FUNCTION_BLOCK FB_Krajalnica_Komunikacja EXTENDS FB_LogowanieBledow_ElementZlozony
VAR_INPUT
END_VAR
VAR_OUTPUT
END_VAR
VAR
END_VAR

METHOD DefinicjaTabeliZdarzen_1031_Niemiecki : BOOL
VAR_INPUT
	arrTablicaDefinicjiZdarzenOpis			: REFERENCE TO ARRAY [1..GVL_LogowanieBledow_Stale.MAX_ILOSC_ZDARZEN] OF DUT_LogowanieBledow_ZdarzenieOpis;

END_VAR
//arrTablicaDefinicjiZdarzenOpis [iStartId+0].sOpis	:= 'DE - TESTOWA WIADOMOSC';
END_METHOD

METHOD DefinicjaTabeliZdarzen_1033_Angielski : BOOL
VAR_INPUT
	arrTablicaDefinicjiZdarzenOpis			: REFERENCE TO ARRAY [1..GVL_LogowanieBledow_Stale.MAX_ILOSC_ZDARZEN] OF DUT_LogowanieBledow_ZdarzenieOpis;

END_VAR
//arrTablicaDefinicjiZdarzenOpis [iStartId+0].sOpis	:= 'EN - TESTOWA WIADOMOSC';
END_METHOD

METHOD DefinicjaTabeliZdarzen_1045_Polski : BOOL
VAR_INPUT
	arrTablicaDefinicjiZdarzenOpis			: REFERENCE TO ARRAY [1..GVL_LogowanieBledow_Stale.MAX_ILOSC_ZDARZEN] OF DUT_LogowanieBledow_ZdarzenieOpis;

END_VAR
//arrTablicaDefinicjiZdarzenOpis [iStartId+0].sOpis	:= 'PL - TESTOWA WIADOMOSC';
END_METHOD

METHOD DefinicjaTabeliZdarzen_Ogolna : BOOL
VAR_INPUT
	arrTablicaDefinicjiZdarzen				: REFERENCE TO ARRAY [1..GVL_LogowanieBledow_Stale.MAX_ILOSC_ZDARZEN] OF DUT_LogowanieBledow_Zdarzenie;
	arrTablicaDefinicjiZdarzenOpis			: REFERENCE TO ARRAY [1..GVL_LogowanieBledow_Stale.MAX_ILOSC_ZDARZEN] OF DUT_LogowanieBledow_ZdarzenieOpis;
	arrTablicaDefinicjiZdarzenStan			: REFERENCE TO ARRAY [1..GVL_LogowanieBledow_Stale.MAX_ILOSC_ZDARZEN] OF DUT_LogowanieBledow_ZdarzenieStan;

	iIdZdarzenia							: REFERENCE TO INT;
	iNrPodzespolu							: INT := 0;
	iNrPodelementu							: INT := 0;
	iNrElementu								: INT := 0;
END_VAR
(*
//testowy blad
	iIdZdarzenia												:= iIdZdarzenia + 1;
	arrTablicaDefinicjiZdarzen [iIdZdarzenia].iIdZdarzenia		:= iIdZdarzenia;
	arrTablicaDefinicjiZdarzen [iIdZdarzenia].byRodzajZdarzenia	:= 3;
	arrTablicaDefinicjiZdarzen [iIdZdarzenia].sKodBledu			:= '0001';
	arrTablicaDefinicjiZdarzen [iIdZdarzenia].sNrKomponentu		:= GenerujNrKomponentu (iNrPodzespolu := iNrPodzespolu, iNrPodelementu := iNrPodelementu, iNrElementu := iNrElementu); 
	arrTablicaDefinicjiZdarzenOpis [iIdZdarzenia].iIdZdarzenia 	:= iIdZdarzenia;
	arrTablicaDefinicjiZdarzenStan [iIdZdarzenia].iIdZdarzenia 	:= iIdZdarzenia;
	arrTablicaDefinicjiZdarzenStan [iIdZdarzenia].bAktywne		:= FALSE;
	*)
END_METHOD

END_FUNCTION_BLOCK

(* stored: Version 1.1.0.1, ProductVersion 3.1.4024.11
   POU FB_Krajalnica_Komunikacja: Id {24ec660a-fdec-41af-bd16-00332dcc9c61}, SpecialFunc None
   Method DefinicjaTabeliZdarzen_1031_Niemiecki: Id {782ca1b3-6969-4262-a0a7-fcec370d5ba6}
   Method DefinicjaTabeliZdarzen_1033_Angielski: Id {9398542a-d901-4a63-a5a2-55dbeb1effe3}
   Method DefinicjaTabeliZdarzen_1045_Polski: Id {7f8f933e-f70b-4985-9665-f7dc640ff2ce}
   Method DefinicjaTabeliZdarzen_Ogolna: Id {060bf940-87c2-490d-800a-aa313bbf9092} *)
